// TwinCAT 3 PLC project VisionLibrary
// ProgramVersion: 3.1.4023.0
// libraries:
//   Tc2_MC2, * (Beckhoff Automation GmbH)
//   Tc2_Standard, * (Beckhoff Automation GmbH)
//   Tc2_System, * (Beckhoff Automation GmbH)
//   Tc3_Module, * (Beckhoff Automation GmbH)
//   VisuDialogs, * (System)
// project tree:
//   DUTs/ SensorToPlc.TcDUT, PlcToSensor.TcDUT, VisionCmd.TcDUT (not stored), VisionState.TcDUT
//   / GlobalTextList.TcGTLO, PlcTask.TcTTO, Visualization Manager.TcVMO (not stored)
//   GVLs/ GVL.TcGVL
//   POUs/ MAIN.TcPOU
//   POUs/VisionBlocks/ SensorFQM.TcPOU
//   VISUs/ HMI.TcVIS
// real-time tasks:
//   TASK PlcTask: cycle T#10ms, priority 20, ADS port 350
// I/O:
//   DEVICE Device 2 (EtherCAT), AmsNetId 10.0.2.15.3.1
//     Term 4 (EK1100) [EK1100 EtherCAT Coupler (2A E-Bus)]
//       Term 5 (EL2008) [EL2008 8Ch. Dig. Output 24V, 0.5A]
//       Term 7 (EL9011) [EL9011 End Terminal]
//     Box 6 (FQ-MS12x-ECT) [FQ-MS12x-ECT]
// variable links:
//   VisionLibrary/VisionLibrary Instance <-> Device 2 (EtherCAT)/Box 6 (FQ-MS12x-ECT)
//     PlcTask Inputs/GVL.FQM.SensorToPlc/VisionDataOutput1 <-> 259th transmit PDO Mapping/Vision Data Output1
//     PlcTask Inputs/GVL.FQM.SensorToPlc/VisionDataOutput2 <-> 259th transmit PDO Mapping/Vision Data Output2
//     PlcTask Inputs/GVL.FQM.SensorToPlc/VisionResponseCode <-> 258th transmit PDO Mapping/Vision Response Code
//     PlcTask Inputs/GVL.FQM.SensorToPlc/VisionResponseData <-> 258th transmit PDO Mapping/Vision Response Data1
//     PlcTask Inputs/GVL.FQM.SensorToPlc/VisionStatusFlag <-> 256th transmit PDO Mapping/Vision Status Flag
//     PlcTask Outputs/GVL.FQM.PlcToSensor/VisionCommand <-> 258th receive PDO Mapping/Vision Command
//     PlcTask Outputs/GVL.FQM.PlcToSensor/VisionControlFlag <-> 256th receive PDO Mapping/SubIndex 001

CONFIGURATION VisionLibrary
    RESOURCE PLC ON TwinCAT3
        TASK PlcTask(INTERVAL := T#10ms, PRIORITY := 20);
        PROGRAM MAIN WITH PlcTask : MAIN;
    END_RESOURCE
END_CONFIGURATION

// ---- DUTs/SensorToPlc.TcDUT
TYPE SensorToPlc :
STRUCT
	VisionStatusFlag AT %I*:DWORD; //Doble Palabra que contiene los bits siguientes
	FLG:BOOL; //Posicion 0
	BUSY:BOOL; //Posicion 1
	READY:BOOL; //Posicion 2
	OR_Jud:BOOL; //Posicion 3
	RUN:BOOL; //Posicion 4
	ERR:BOOL; //Posicion 15
	GATE:BOOL; //Posicion 16
	
	VisionResponseCode AT %I*:DWORD;
	VisionResponseData AT %I*:DWORD;
	
	//Lecturas desde el sensor
	VisionDataOutput1 AT %I*:REAL;
	VisionDataOutput2 AT %I*:REAL;
	VisionDataOutput3 AT %I*:REAL;
	VisionDataOutput4 AT %I*:REAL;
	VisionDataOutput5 AT %I*:REAL;
	VisionDataOutput6 AT %I*:REAL;
	VisionDataOutput7 AT %I*:REAL;
	VisionDataOutput8 AT %I*:REAL;
	
END_STRUCT
END_TYPE

// ---- DUTs/PlcToSensor.TcDUT
TYPE PlcToSensor :
STRUCT
	VisionCommand AT %Q*:DWORD;
	VisionControlFlag AT %Q*:DWORD;
	EXE:BOOL;
	TRIG:BOOL;
	DSA:BOOL;
	ERCLR:BOOL;
END_STRUCT
END_TYPE

// ---- DUTs/VisionState.TcDUT
{attribute 'qualified_only'}
{attribute 'strict'}
TYPE VisionState :
(
	Error := 000,
	StandStill := 010,
	Continuous := 020,
	Discrete := 030
);
END_TYPE

// ---- GVLs/GVL.TcGVL
{attribute 'qualified_only'}
VAR_GLOBAL
	FQM:SensorFQM;
END_VAR

// ---- POUs/MAIN.TcPOU
PROGRAM MAIN
VAR
	Single:BOOL;
	Reset:bool;
	foto: BOOL;
	HaveResult:BOOL;
	Resultado: ARRAY [0..7] OF REAL;
END_VAR


GVL.FQM.SingleShot(Enable:=Single,Execute:=foto,Measurement => HaveResult, Results => Resultado);
GVL.FQM();

END_PROGRAM

// ---- POUs/VisionBlocks/SensorFQM.TcPOU
FUNCTION_BLOCK SensorFQM
VAR_INPUT
END_VAR
VAR_OUTPUT
END_VAR
VAR_IN_OUT
	
END_VAR
VAR
	State:INT:= 10;
	SensorToPlc AT %I*:SensorToPlc;
	PlcToSensor AT %Q*:PlcToSensor;
	KeepAliveTimer:TON;
	
	RExec:R_TRIG;
	NextCycleResetFlags:BOOL;
	
	
	//Single measurement
	RequestSingle:BOOL;
	TakePhoto:BOOL;
	TakePhotoFlag:R_TRIG;
	MeasurementTimer:TON;
	MeasureTime:TIME;
	
	LastResult:INT:=0;//0-Null, 1-Ok, 2-NG
	//Error Management
	RequestErrorCode:BOOL;
	LastError:DWORD;
	Resultado:REAL;
END_VAR
VAR CONSTANT
	KeepAliveBit:INT:=24;
END_VAR

// Preparing Inputs
SensorToPlc.FLG:= SensorToPlc.VisionStatusFlag.0;
SensorToPlc.BUSY:= SensorToPlc.VisionStatusFlag.1;
SensorToPlc.READY:= SensorToPlc.VisionStatusFlag.2;
SensorToPlc.OR_Jud:= SensorToPlc.VisionStatusFlag.3;
SensorToPlc.RUN:= SensorToPlc.VisionStatusFlag.4;
SensorToPlc.ERR:= SensorToPlc.VisionStatusFlag.15;
SensorToPlc.GATE:= SensorToPlc.VisionStatusFlag.16;
//Change a bit every 500ms as Keep Alive bit
KeepAliveTimer(in:=NOT KeepAliveTimer.Q, pt:=T#500MS);
IF KeepAliveTimer.Q THEN
	PlcToSensor.VisionControlFlag.24:= NOT PlcToSensor.VisionControlFlag.24;
END_IF

//State machine
CASE State OF
	000: //Error
		PlcToSensor.ERCLR:=FALSE;
		IF NOT SensorToPlc.ERR THEN
			State := 010;
		ELSE
			State := 001;
		END_IF
			
	001: //Checking errors
		//TODO: Revisar
		IF SensorToPlc.FLG THEN
			PlcToSensor.EXE:=FALSE;
			LastError:= SensorToPlc.VisionResponseCode;
			PlcToSensor.ERCLR:=TRUE;
		END_IF
	010: //StandStill
		IF RequestSingle THEN
			PrepareCommand(VisionCmd.StartSingle);
			PlcToSensor.EXE:=TRUE;
			State := 011;
		END_IF
		
	011: //Switching to Single
		IF SensorToPlc.FLG THEN
			PlcToSensor.EXE := FALSE;
			State := 030;
			LastResult:=0;
		END_IF
	030: // Single Measurement Ready
		
		IF TakePhoto THEN
			//Take photo and request
			PlcToSensor.TRIG:=TRUE;
			PlcToSensor.DSA:=TRUE;
			MeasurementTimer(in:=FALSE);
			MeasurementTimer(in:=TRUE, pt:=T#60s);
			State := 31;
		END_IF
		IF NOT RequestSingle THEN
			State := 010;
		END_IF
		IF SensorToPlc.ERR THEN
			State := 001;
			PrepareCommand(Command:= VisionCmd.GetLatestError);
			PlcToSensor.EXE := TRUE;
		END_IF
	031: // Single Measurement Taking photo
		MeasurementTimer(in:=TRUE);
		IF SensorToPLC.GATE THEN
			IF SensorToPlc.OR_Jud THEN
				LastResult:=2;
			ELSE
				LastResult:=1;
			END_IF	
			Resultado:= SensorToPlc.VisionDataOutput1;
			MeasureTime:=MeasurementTimer.ET;
			MeasurementTimer(in:=FALSE);
			State := 030;
			PlcToSensor.TRIG:=FALSE;
			PlcToSensor.DSA:=FALSE;
		END_IF
		IF SensorToPLC.ERR THEN
			State := 001;
		END_IF
END_CASE

//Update Flag Bits into DWORD
PlcToSensor.VisionControlFlag.0:= PlcToSensor.EXE;
PlcToSensor.VisionControlFlag.1:= PlcToSensor.TRIG;
PlcToSensor.VisionControlFlag.15:= PlcToSensor.ERCLR;
PlcToSensor.VisionControlFlag.16:= PlcToSensor.DSA;

METHOD PRIVATE PrepareCommand
VAR_INPUT
	Command:VisionCmd;
END_VAR
VAR
	
END_VAR
CASE Command OF
	VisionCmd.StartSingle: PlcToSensor.VisionCommand:= 16#00101010;
	VisionCmd.StartContinuous: PlcToSensor.VisionCommand:= 16#00101020;
	VisionCmd.StopContinuous: PlcToSensor.VisionCommand:= 16#00101030;
	VisionCmd.ClearValues: PlcToSensor.VisionCommand:= 16#00102010;
	VisionCmd.ClearDataOutputBuffer: PlcToSensor.VisionCommand:= 16#00102020;
	VisionCmd.Reset: PlcToSensor.VisionCommand:= 16#0010F010;
	VisionCmd.GetLatestError: PlcToSensor.VisionCommand:= 16#00205000;
END_CASE
END_METHOD

METHOD PUBLIC SingleShot : BOOL
VAR_INPUT
	Enable:BOOL;
	Execute:BOOL;
END_VAR
VAR_OUTPUT
	Active:BOOL;
	Measurement:BOOL;
	Ok:BOOL;
	Ng:BOOL;
	Results: ARRAY [0..7] OF REAL;
END_VAR
IF Enable THEN
	RequestSingle:=TRUE;
ELSE
	RequestSingle:=FALSE;
END_IF

TakePhotoFlag(clk:= Execute);
IF State = 030 THEN
	Active:=TRUE;
	IF TakePhotoFlag.Q THEN
		TakePhoto:=TRUE;
		Ok:=FALSE;
		Ng:=FALSE;
	END_IF
	CASE LastResult OF
		0: Ok:=FALSE; Ng:=FALSE; Measurement:=FALSE;
		1: Ok:=TRUE; Ng:=FALSE; Measurement:=TRUE;
		2: Ok:=FALSE; Ng:=TRUE; Measurement:= TRUE;
	END_CASE
	Results[0]:= SensorToPlc.VisionDataOutput1;
	Results[1]:= SensorToPlc.VisionDataOutput2;
	Results[2]:= SensorToPlc.VisionDataOutput3;
	Results[3]:= SensorToPlc.VisionDataOutput4;
	Results[4]:= SensorToPlc.VisionDataOutput5;
	Results[5]:= SensorToPlc.VisionDataOutput6;
	Results[6]:= SensorToPlc.VisionDataOutput7;
	Results[7]:= SensorToPlc.VisionDataOutput8;
ELSIF State = 031 THEN
	TakePhoto:=FALSE;
END_IF
END_METHOD

END_FUNCTION_BLOCK

// ---- GlobalTextList.TcGTLO
TEXTLIST GlobalTextList
  512 = '%s'
  831 = 'Comando'
  740 = 'd'
  761 = 'Distancia'
  101 = 'EndContinuous'
  116 = 'Foto'
  781 = 'Iniciar Single \nMeasurement'
  856 = 'Iniciar Single Measurement'
  122 = 'Medida1'
  84 = 'Prueba'
  226 = 'Resultados'
  619 = 'Start Continuous'
  922 = 'StartContinuous'
  315 = 'StartSingle'
  64 = 'StartSingle:  10100010'
  393 = 'StartSingle:  10100010\n'
  736 = 'StartSingle:  10100010\nStartCont: 00101020\nStopCont: 10300010\nGetLastError: 00205000'
  592 = 'StartSingle:  10100010\\n\\r'
  330 = 'VarAux'
END_TEXTLIST

// ---- VISUs/HMI.TcVIS
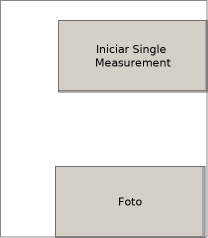
VISUALIZATION HMI  // 208x238
    Button (55,166 150x72), "Foto"
        tap MAIN.foto
    Button (58,20 150x72), "Iniciar Single Measurement"
        toggle MAIN.Single
END_VISUALIZATION
